// TIA Portal V21 export
FUNCTION_BLOCK "FB302"   // FB302, LAD
TITLE = FB302
{ S7_Optimized_Access := 'TRUE' }
AUTHOR : PRECISE
FAMILY : PRECISE
// MIXING
// stored: AutoNumber false, MemoryReserve 100, SetENOAutomatically false
   VAR_INPUT
      Enable : Bool;
      Disable : Bool;
      Fault : Bool;
      SecPulse : Bool;
      AlwaysTrue : Bool;
      StartConfirmationPopupSel : Bool;   // StartConfirmationPopupSel: 0-NO/1-YES
      EndConfirmationPopupSel : Bool;   // EndConfirmationPopupSel: 0-NO/1-YES
      MixingModeSel : Int;   // Mixing Mode Selection: 0-Auto/1-Manual
      MixerTypeSel : Int;   // Mixer Type Selection: 0-MM/1-USM/2-HSM/3-BP/4-ANCHOR
      MixingTimeBaseSel : Bool;   // Mixing Time Base Selection: 0-second/1-minute
      MixingTimeMin : Int := 1;   // For Mixing Mode Selection: 0-Auto & Mixing Time Base Selection: 1-minute
      MixingTimeSec : Int := 30;   // For Mixing Mode Selection: 0-Auto & Mixing Time Base Selection: 0-second
      MixingSpeed : Real := 100.0;
   END_VAR
   VAR_OUTPUT
      MixerCmd : Bool;
      WaterInletValve : Bool;
      StartConfirmationPopup : Bool;   // For Start Confirmation Popup Selection: Yes
      EndConfirmationPopup : Bool;   // For End Confirmation Popup Selection: Yes
      ManualPopup : Bool;   // For Mixing Mode Selection: 1-Manual
      MixingTimeMinPV : DInt;   // For Mixing Mode Selection: 0-Auto
      MixingTimeSecPV : DInt;   // For Mixing Mode Selection: 0-Auto
      MixingSpeedPV : Real;
      PrintTrigger : Bool;
      PrintWord : Int;
      PrintStatus : String[50];
   END_VAR
   VAR_IN_OUT
      Start : Bool;
      Stop : Bool;
      Reset : Bool;
      StartConfirmationAck : Bool;   // For Start Confirmation Popup Selection: Yes
      EndConfirmationAck : Bool;   // For End Confirmation Popup Selection: Yes
      ManualAck : Bool;   // For Mixing Mode Selection: 1-Manual
      Cp01Fsc : Bool;
      SpareBtn2 : Bool;
      Running : Bool;
      Selected : Bool;
      Paused : Bool;
      StartConfirmationPopupTemp : Bool;   // For Start Confirmation Popup Selection: Yes
      EndConfirmationPopupTemp : Bool;   // For End Confirmation Popup Selection: Yes
      ManualPopupTemp : Bool;   // For Mixing Mode Selection: 1-Manual
      MixingStarted : Bool;
      MixingOver : Bool;
   END_VAR
   VAR
      PrintTriggerTemp : Bool;
      RE1 : Bool;
      RE2 : Bool;
      RE3 : Bool;
      RE4 : Bool;
      RE5 : Bool;
      RE6 : Bool;
      RE7 : Bool;
      MixingTimer : "FB101";
      PrintTriggerResetTimer { S7_SetPoint := 'True'} : TON_TIME;
      BtnResetTimer { S7_SetPoint := 'True'} : TON_TIME;
   END_VAR
   VAR_TEMP
      STATUS1 : String[40];
      STATUS2 : String[40];
      STATUS3 : String[40];
      STATUS4 : String[40];
      STATUS5 : String[40];
   END_VAR
   VAR_TEMP   // added for the SCL form of the ladder/FBD networks
      _w1 : Bool;
      _w2 : Bool;
      _w3 : Bool;
      _w4 : Bool;
      _w5 : Bool;
   END_VAR
BEGIN

REGION Network 1: Running
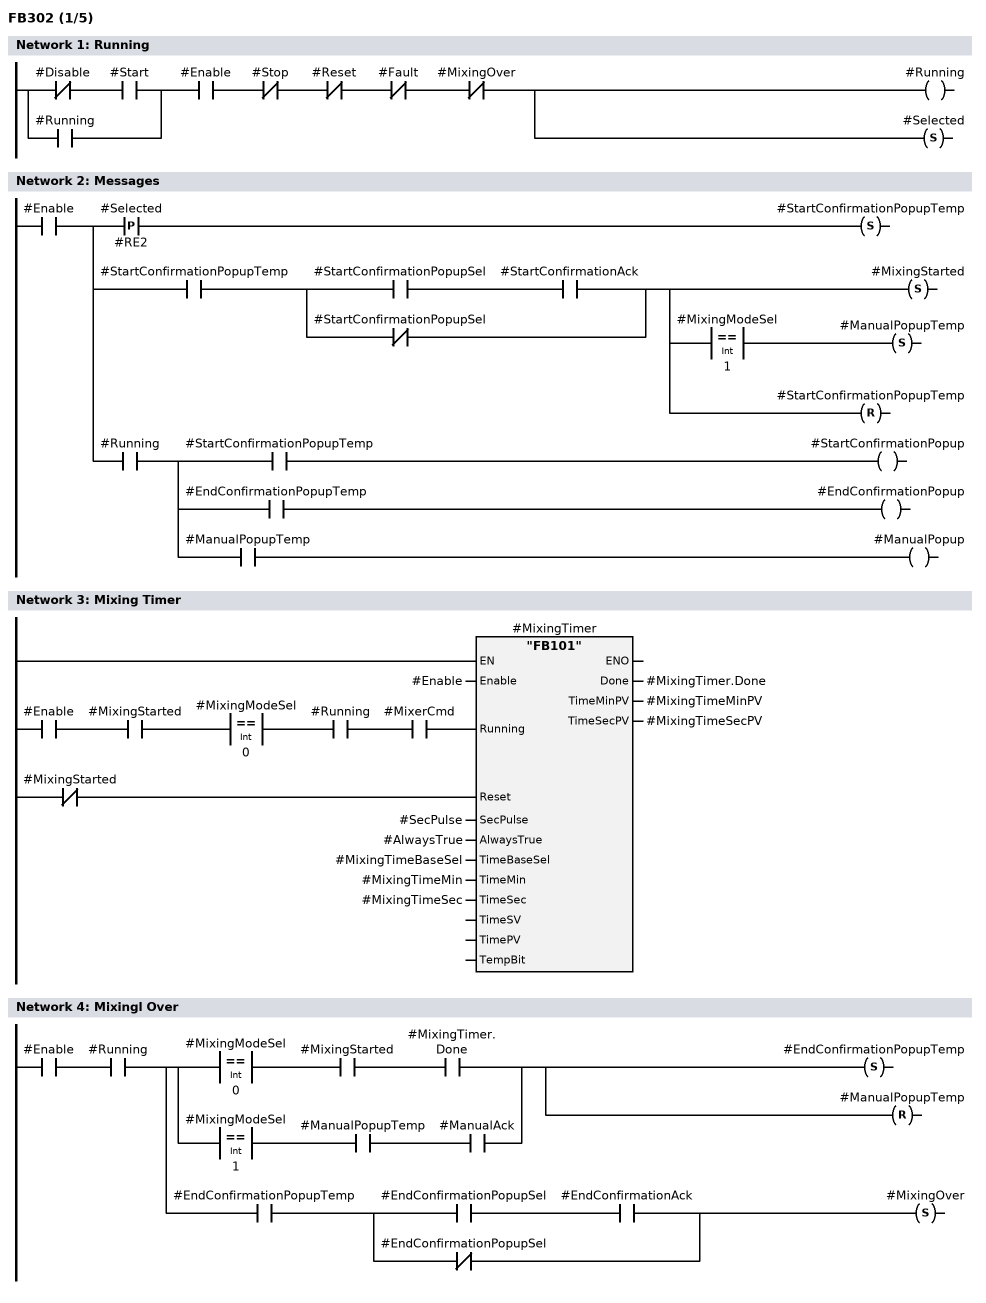
   RUNG wire#powerrail
      I_Contact( #Disable )
      Contact( #Start )
      wire#w1
      Contact( #Enable )
      I_Contact( #Stop )
      I_Contact( #Reset )
      I_Contact( #Fault )
      I_Contact( #MixingOver )
      wire#w2
      Coil( #Running )
   END_RUNG
   RUNG wire#powerrail
      Contact( #Running )
   END_RUNG wire#w1
   RUNG wire#w2
      S_Coil( #Selected )
   END_RUNG
   // the same network as SCL:
   #Running := ((NOT #Disable AND #Start) OR #Running) AND #Enable AND NOT #Stop AND NOT #Reset AND NOT #Fault AND NOT #MixingOver;
   IF #Running THEN #Selected := TRUE; END_IF;
END_REGION

REGION Network 2: Messages
   RUNG wire#powerrail
      Contact( #Enable )
      wire#w1
      P_Contact(operand := #Selected, bit := #RE2)
      S_Coil( #StartConfirmationPopupTemp )
   END_RUNG
   RUNG wire#w1
      Contact( #StartConfirmationPopupTemp )
      wire#w2
      Contact( #StartConfirmationPopupSel )
      Contact( #StartConfirmationAck )
      wire#w3
      S_Coil( #MixingStarted )
   END_RUNG
   RUNG wire#w2
      I_Contact( #StartConfirmationPopupSel )
   END_RUNG wire#w3
   RUNG wire#w3
      { S7_Templates := "SrcType := Int" } EQ_Contact(in1 := #MixingModeSel, in2 := 1)
      S_Coil( #ManualPopupTemp )
   END_RUNG
   RUNG wire#w3
      R_Coil( #StartConfirmationPopupTemp )
   END_RUNG
   RUNG wire#w1
      Contact( #Running )
      wire#w4
      Contact( #StartConfirmationPopupTemp )
      Coil( #StartConfirmationPopup )
   END_RUNG
   RUNG wire#w4
      Contact( #EndConfirmationPopupTemp )
      Coil( #EndConfirmationPopup )
   END_RUNG
   RUNG wire#w4
      Contact( #ManualPopupTemp )
      Coil( #ManualPopup )
   END_RUNG
   // the same network as SCL:
   #_w1 := #Enable AND #Selected AND NOT #RE2;   // rising edge of #Selected
   #RE2 := #Selected;
   IF #_w1 THEN #StartConfirmationPopupTemp := TRUE; END_IF;
   #_w2 := #Enable AND #StartConfirmationPopupTemp AND ((#StartConfirmationPopupSel AND #StartConfirmationAck) OR NOT #StartConfirmationPopupSel);
   IF #_w2 THEN #MixingStarted := TRUE; END_IF;
   IF #_w2 AND (#MixingModeSel = 1) THEN #ManualPopupTemp := TRUE; END_IF;
   IF #_w2 THEN #StartConfirmationPopupTemp := FALSE; END_IF;
   #_w3 := #Enable AND #Running;
   #StartConfirmationPopup := #_w3 AND #StartConfirmationPopupTemp;
   #EndConfirmationPopup := #_w3 AND #EndConfirmationPopupTemp;
   #ManualPopup := #_w3 AND #ManualPopupTemp;
END_REGION

REGION Network 3: Mixing Timer
   RUNG wire#powerrail
      #MixingTimer(Running := wire#w1, Reset := wire#w2, Enable := #Enable, SecPulse := #SecPulse, AlwaysTrue := #AlwaysTrue, TimeBaseSel := #MixingTimeBaseSel, TimeMin := #MixingTimeMin, TimeSec := #MixingTimeSec, TimeSV :=, TimePV :=, TempBit :=, Done => #MixingTimer.Done, TimeMinPV => #MixingTimeMinPV, TimeSecPV => #MixingTimeSecPV)
   END_RUNG
   RUNG wire#powerrail
      Contact( #Enable )
      Contact( #MixingStarted )
      { S7_Templates := "SrcType := Int" } EQ_Contact(in1 := #MixingModeSel, in2 := 0)
      Contact( #Running )
      Contact( #MixerCmd )
   END_RUNG wire#w1
   RUNG wire#powerrail
      I_Contact( #MixingStarted )
   END_RUNG wire#w2
   // the same network as SCL:
   #MixingTimer(Enable := #Enable,   // "FB101"
                Running := #Enable AND #MixingStarted AND (#MixingModeSel = 0) AND #Running AND #MixerCmd,
                Reset := NOT #MixingStarted,
                SecPulse := #SecPulse,
                AlwaysTrue := #AlwaysTrue,
                TimeBaseSel := #MixingTimeBaseSel,
                TimeMin := #MixingTimeMin,
                TimeSec := #MixingTimeSec,
                Done => #MixingTimer.Done,
                TimeMinPV => #MixingTimeMinPV,
                TimeSecPV => #MixingTimeSecPV);
END_REGION

REGION Network 4: Mixingl Over
   RUNG wire#powerrail
      Contact( #Enable )
      Contact( #Running )
      wire#w1
      { S7_Templates := "SrcType := Int" } EQ_Contact(in1 := #MixingModeSel, in2 := 0)
      Contact( #MixingStarted )
      Contact( #MixingTimer.Done )
      wire#w2
      S_Coil( #EndConfirmationPopupTemp )
   END_RUNG
   RUNG wire#w1
      { S7_Templates := "SrcType := Int" } EQ_Contact(in1 := #MixingModeSel, in2 := 1)
      Contact( #ManualPopupTemp )
      Contact( #ManualAck )
   END_RUNG wire#w2
   RUNG wire#w2
      R_Coil( #ManualPopupTemp )
   END_RUNG
   RUNG wire#w1
      Contact( #EndConfirmationPopupTemp )
      wire#w3
      Contact( #EndConfirmationPopupSel )
      Contact( #EndConfirmationAck )
      wire#w4
      S_Coil( #MixingOver )
   END_RUNG
   RUNG wire#w3
      I_Contact( #EndConfirmationPopupSel )
   END_RUNG wire#w4
   // the same network as SCL:
   #_w1 := #Enable AND #Running;
   IF #_w1 AND (((#MixingModeSel = 0) AND #MixingStarted AND #MixingTimer.Done) OR ((#MixingModeSel = 1) AND #ManualPopupTemp AND #ManualAck)) THEN
       #EndConfirmationPopupTemp := TRUE;
       #ManualPopupTemp := FALSE;
   END_IF;
   IF #_w1 AND #EndConfirmationPopupTemp AND ((#EndConfirmationPopupSel AND #EndConfirmationAck) OR NOT #EndConfirmationPopupSel) THEN
       #MixingOver := TRUE;
   END_IF;
END_REGION

REGION Network 5: Output On
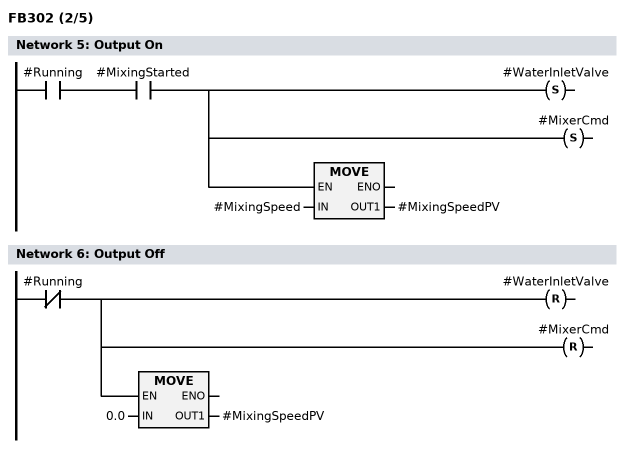
   RUNG wire#powerrail
      Contact( #Running )
      Contact( #MixingStarted )
      wire#w1
      S_Coil( #WaterInletValve )
   END_RUNG
   RUNG wire#w1
      S_Coil( #MixerCmd )
   END_RUNG
   RUNG wire#w1
      Move(in := #MixingSpeed, out1 => #MixingSpeedPV)
   END_RUNG
   // the same network as SCL:
   IF #Running AND #MixingStarted THEN
       #WaterInletValve := TRUE;
       #MixerCmd := TRUE;
       #MixingSpeedPV := #MixingSpeed;
   END_IF;
END_REGION

REGION Network 6: Output Off
   RUNG wire#powerrail
      I_Contact( #Running )
      wire#w1
      R_Coil( #WaterInletValve )
   END_RUNG
   RUNG wire#w1
      R_Coil( #MixerCmd )
   END_RUNG
   RUNG wire#w1
      Move(in := 0.0, out1 => #MixingSpeedPV)
   END_RUNG
   // the same network as SCL:
   IF NOT #Running THEN
       #WaterInletValve := FALSE;
       #MixerCmd := FALSE;
       #MixingSpeedPV := 0.0;
   END_IF;
END_REGION

REGION Network 7: Event Status
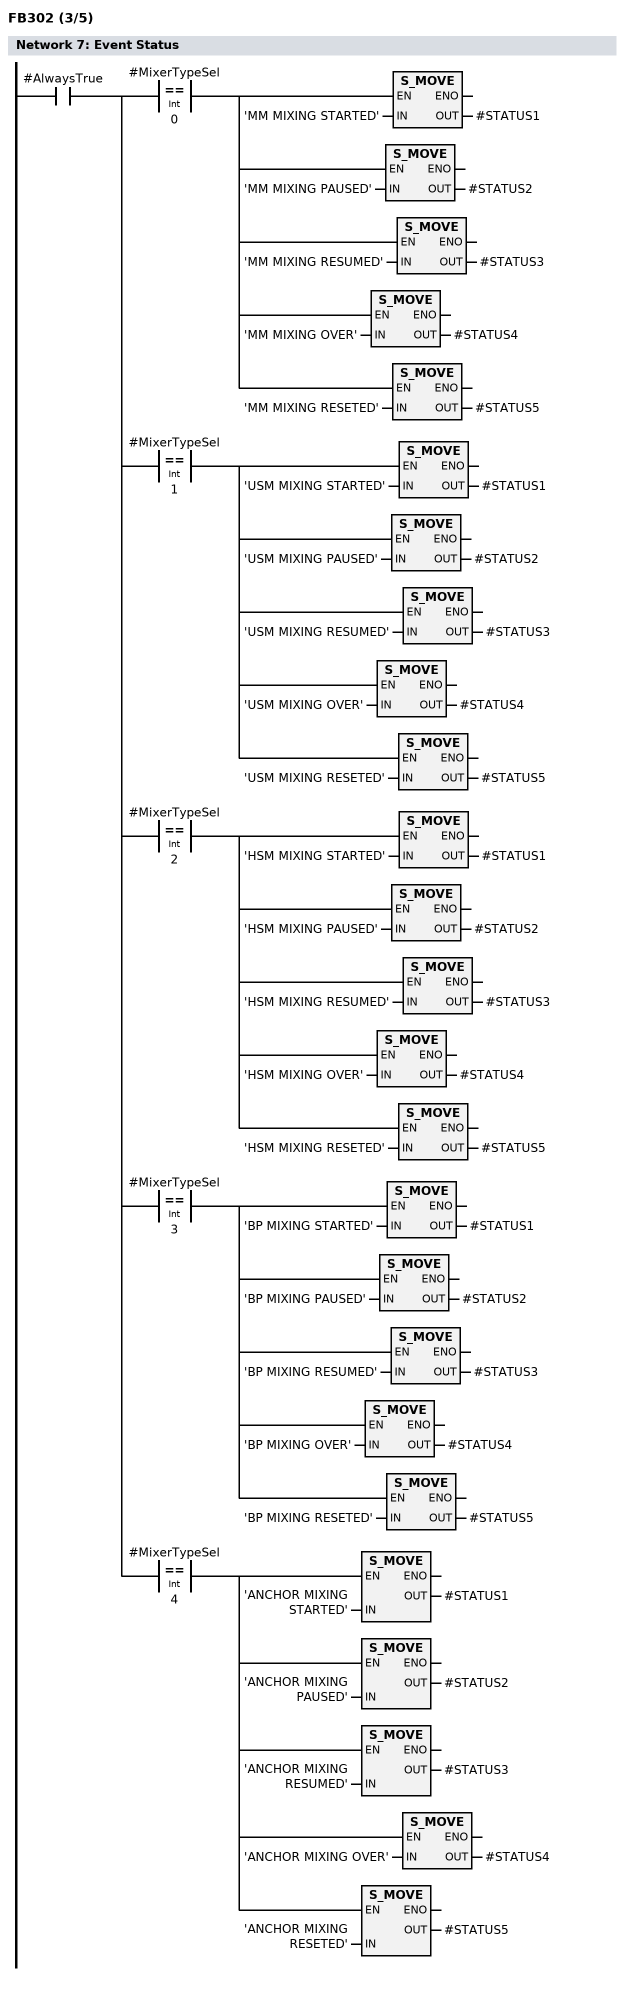
   RUNG wire#powerrail
      Contact( #AlwaysTrue )
      wire#w1
      { S7_Templates := "SrcType := Int" } EQ_Contact(in1 := #MixerTypeSel, in2 := 0)
      wire#w2
      S_Move(in := 'MM MIXING STARTED', out => #STATUS1)
   END_RUNG
   RUNG wire#w2
      S_Move(in := 'MM MIXING PAUSED', out => #STATUS2)
   END_RUNG
   RUNG wire#w2
      S_Move(in := 'MM MIXING RESUMED', out => #STATUS3)
   END_RUNG
   RUNG wire#w2
      S_Move(in := 'MM MIXING OVER', out => #STATUS4)
   END_RUNG
   RUNG wire#w2
      S_Move(in := 'MM MIXING RESETED', out => #STATUS5)
   END_RUNG
   RUNG wire#w1
      { S7_Templates := "SrcType := Int" } EQ_Contact(in1 := #MixerTypeSel, in2 := 1)
      wire#w3
      S_Move(in := 'USM MIXING STARTED', out => #STATUS1)
   END_RUNG
   RUNG wire#w3
      S_Move(in := 'USM MIXING PAUSED', out => #STATUS2)
   END_RUNG
   RUNG wire#w3
      S_Move(in := 'USM MIXING RESUMED', out => #STATUS3)
   END_RUNG
   RUNG wire#w3
      S_Move(in := 'USM MIXING OVER', out => #STATUS4)
   END_RUNG
   RUNG wire#w3
      S_Move(in := 'USM MIXING RESETED', out => #STATUS5)
   END_RUNG
   RUNG wire#w1
      { S7_Templates := "SrcType := Int" } EQ_Contact(in1 := #MixerTypeSel, in2 := 2)
      wire#w4
      S_Move(in := 'HSM MIXING STARTED', out => #STATUS1)
   END_RUNG
   RUNG wire#w4
      S_Move(in := 'HSM MIXING PAUSED', out => #STATUS2)
   END_RUNG
   RUNG wire#w4
      S_Move(in := 'HSM MIXING RESUMED', out => #STATUS3)
   END_RUNG
   RUNG wire#w4
      S_Move(in := 'HSM MIXING OVER', out => #STATUS4)
   END_RUNG
   RUNG wire#w4
      S_Move(in := 'HSM MIXING RESETED', out => #STATUS5)
   END_RUNG
   RUNG wire#w1
      { S7_Templates := "SrcType := Int" } EQ_Contact(in1 := #MixerTypeSel, in2 := 3)
      wire#w5
      S_Move(in := 'BP MIXING STARTED', out => #STATUS1)
   END_RUNG
   RUNG wire#w5
      S_Move(in := 'BP MIXING PAUSED', out => #STATUS2)
   END_RUNG
   RUNG wire#w5
      S_Move(in := 'BP MIXING RESUMED', out => #STATUS3)
   END_RUNG
   RUNG wire#w5
      S_Move(in := 'BP MIXING OVER', out => #STATUS4)
   END_RUNG
   RUNG wire#w5
      S_Move(in := 'BP MIXING RESETED', out => #STATUS5)
   END_RUNG
   RUNG wire#w1
      { S7_Templates := "SrcType := Int" } EQ_Contact(in1 := #MixerTypeSel, in2 := 4)
      wire#w6
      S_Move(in := 'ANCHOR MIXING STARTED', out => #STATUS1)
   END_RUNG
   RUNG wire#w6
      S_Move(in := 'ANCHOR MIXING PAUSED', out => #STATUS2)
   END_RUNG
   RUNG wire#w6
      S_Move(in := 'ANCHOR MIXING RESUMED', out => #STATUS3)
   END_RUNG
   RUNG wire#w6
      S_Move(in := 'ANCHOR MIXING OVER', out => #STATUS4)
   END_RUNG
   RUNG wire#w6
      S_Move(in := 'ANCHOR MIXING RESETED', out => #STATUS5)
   END_RUNG
   // the same network as SCL:
   IF #AlwaysTrue AND (#MixerTypeSel = 0) THEN
       #STATUS1 := 'MM MIXING STARTED';
       #STATUS2 := 'MM MIXING PAUSED';
       #STATUS3 := 'MM MIXING RESUMED';
       #STATUS4 := 'MM MIXING OVER';
       #STATUS5 := 'MM MIXING RESETED';
   END_IF;
   IF #AlwaysTrue AND (#MixerTypeSel = 1) THEN
       #STATUS1 := 'USM MIXING STARTED';
       #STATUS2 := 'USM MIXING PAUSED';
       #STATUS3 := 'USM MIXING RESUMED';
       #STATUS4 := 'USM MIXING OVER';
       #STATUS5 := 'USM MIXING RESETED';
   END_IF;
   IF #AlwaysTrue AND (#MixerTypeSel = 2) THEN
       #STATUS1 := 'HSM MIXING STARTED';
       #STATUS2 := 'HSM MIXING PAUSED';
       #STATUS3 := 'HSM MIXING RESUMED';
       #STATUS4 := 'HSM MIXING OVER';
       #STATUS5 := 'HSM MIXING RESETED';
   END_IF;
   IF #AlwaysTrue AND (#MixerTypeSel = 3) THEN
       #STATUS1 := 'BP MIXING STARTED';
       #STATUS2 := 'BP MIXING PAUSED';
       #STATUS3 := 'BP MIXING RESUMED';
       #STATUS4 := 'BP MIXING OVER';
       #STATUS5 := 'BP MIXING RESETED';
   END_IF;
   IF #AlwaysTrue AND (#MixerTypeSel = 4) THEN
       #STATUS1 := 'ANCHOR MIXING STARTED';
       #STATUS2 := 'ANCHOR MIXING PAUSED';
       #STATUS3 := 'ANCHOR MIXING RESUMED';
       #STATUS4 := 'ANCHOR MIXING OVER';
       #STATUS5 := 'ANCHOR MIXING RESETED';
   END_IF;
END_REGION

REGION Network 8: Print Logic
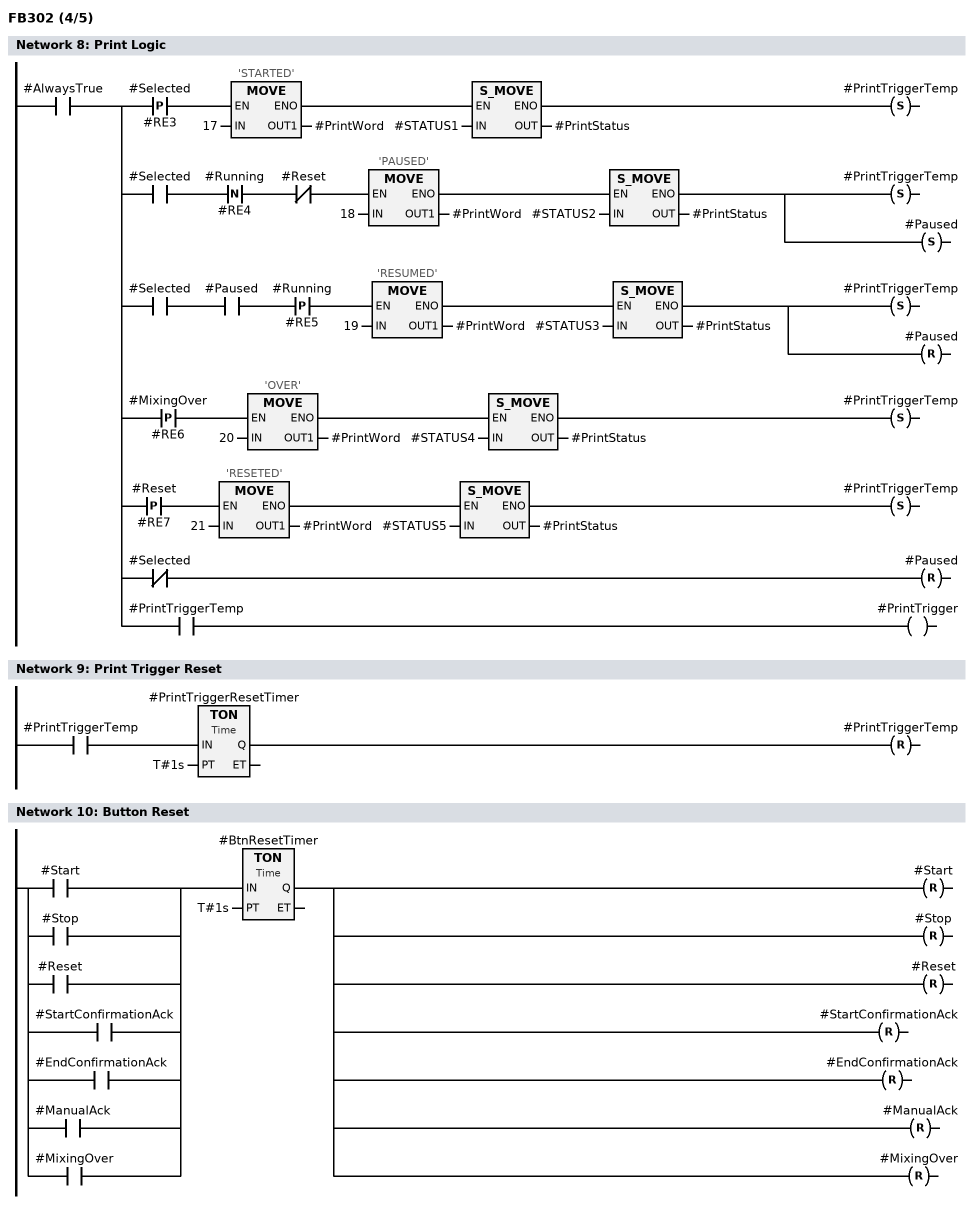
   RUNG wire#powerrail
      Contact( #AlwaysTrue )
      wire#w1
      P_Contact(operand := #Selected, bit := #RE3)
      { S7_GenerateENO := "TRUE" } Move(in := 17, out1 => #PrintWord)   // 'STARTED'
      S_Move(in := #STATUS1, out => #PrintStatus)
      S_Coil( #PrintTriggerTemp )
   END_RUNG
   RUNG wire#w1
      Contact( #Selected )
      N_Contact(operand := #Running, bit := #RE4)
      I_Contact( #Reset )
      { S7_GenerateENO := "TRUE" } Move(in := 18, out1 => #PrintWord)   // 'PAUSED'
      S_Move(in := #STATUS2, out => #PrintStatus)
      wire#w2
      S_Coil( #PrintTriggerTemp )
   END_RUNG
   RUNG wire#w2
      S_Coil( #Paused )
   END_RUNG
   RUNG wire#w1
      Contact( #Selected )
      Contact( #Paused )
      P_Contact(operand := #Running, bit := #RE5)
      { S7_GenerateENO := "TRUE" } Move(in := 19, out1 => #PrintWord)   // 'RESUMED'
      S_Move(in := #STATUS3, out => #PrintStatus)
      wire#w3
      S_Coil( #PrintTriggerTemp )
   END_RUNG
   RUNG wire#w3
      R_Coil( #Paused )
   END_RUNG
   RUNG wire#w1
      P_Contact(operand := #MixingOver, bit := #RE6)
      { S7_GenerateENO := "TRUE" } Move(in := 20, out1 => #PrintWord)   // 'OVER'
      S_Move(in := #STATUS4, out => #PrintStatus)
      S_Coil( #PrintTriggerTemp )
   END_RUNG
   RUNG wire#w1
      P_Contact(operand := #Reset, bit := #RE7)
      { S7_GenerateENO := "TRUE" } Move(in := 21, out1 => #PrintWord)   // 'RESETED'
      S_Move(in := #STATUS5, out => #PrintStatus)
      S_Coil( #PrintTriggerTemp )
   END_RUNG
   RUNG wire#w1
      I_Contact( #Selected )
      R_Coil( #Paused )
   END_RUNG
   RUNG wire#w1
      Contact( #PrintTriggerTemp )
      Coil( #PrintTrigger )
   END_RUNG
   // the same network as SCL:
   // ENO of a box is taken as its EN; it also drops when the box reports an error
   #_w1 := #AlwaysTrue AND #Selected AND NOT #RE3;   // rising edge of #Selected
   #RE3 := #Selected;
   IF #_w1 THEN
       #PrintWord := 17;   // 'STARTED'
       #PrintStatus := #STATUS1;
       #PrintTriggerTemp := TRUE;
   END_IF;
   #_w2 := #AlwaysTrue AND #Selected AND NOT #Running AND #RE4;   // falling edge of #Running
   #RE4 := #Running;
   IF #_w2 AND NOT #Reset THEN
       #PrintWord := 18;   // 'PAUSED'
       #PrintStatus := #STATUS2;
       #PrintTriggerTemp := TRUE;
       #Paused := TRUE;
   END_IF;
   #_w3 := #AlwaysTrue AND #Selected AND #Paused AND #Running AND NOT #RE5;   // rising edge of #Running
   #RE5 := #Running;
   IF #_w3 THEN
       #PrintWord := 19;   // 'RESUMED'
       #PrintStatus := #STATUS3;
       #PrintTriggerTemp := TRUE;
       #Paused := FALSE;
   END_IF;
   #_w4 := #AlwaysTrue AND #MixingOver AND NOT #RE6;   // rising edge of #MixingOver
   #RE6 := #MixingOver;
   IF #_w4 THEN
       #PrintWord := 20;   // 'OVER'
       #PrintStatus := #STATUS4;
       #PrintTriggerTemp := TRUE;
   END_IF;
   #_w5 := #AlwaysTrue AND #Reset AND NOT #RE7;   // rising edge of #Reset
   #RE7 := #Reset;
   IF #_w5 THEN
       #PrintWord := 21;   // 'RESETED'
       #PrintStatus := #STATUS5;
       #PrintTriggerTemp := TRUE;
   END_IF;
   IF #AlwaysTrue AND NOT #Selected THEN #Paused := FALSE; END_IF;
   #PrintTrigger := #AlwaysTrue AND #PrintTriggerTemp;
END_REGION

REGION Network 9: Print Trigger Reset
   RUNG wire#powerrail
      Contact( #PrintTriggerTemp )
      { S7_Templates := "time_type := Time" } #PrintTriggerResetTimer.TON(pt := T#1s, et =>)
      R_Coil( #PrintTriggerTemp )
   END_RUNG
   // the same network as SCL:
   #PrintTriggerResetTimer(IN := #PrintTriggerTemp, PT := T#1s);   // TON
   IF #PrintTriggerResetTimer.Q THEN #PrintTriggerTemp := FALSE; END_IF;
END_REGION

REGION Network 10: Button Reset
   RUNG wire#powerrail
      Contact( #Start )
      wire#w1
      { S7_Templates := "time_type := Time" } #BtnResetTimer.TON(pt := T#1s, et =>)
      wire#w2
      R_Coil( #Start )
   END_RUNG
   RUNG wire#powerrail
      Contact( #Stop )
   END_RUNG wire#w1
   RUNG wire#powerrail
      Contact( #Reset )
   END_RUNG wire#w1
   RUNG wire#powerrail
      Contact( #StartConfirmationAck )
   END_RUNG wire#w1
   RUNG wire#powerrail
      Contact( #EndConfirmationAck )
   END_RUNG wire#w1
   RUNG wire#powerrail
      Contact( #ManualAck )
   END_RUNG wire#w1
   RUNG wire#powerrail
      Contact( #MixingOver )
   END_RUNG wire#w1
   RUNG wire#w2
      R_Coil( #Stop )
   END_RUNG
   RUNG wire#w2
      R_Coil( #Reset )
   END_RUNG
   RUNG wire#w2
      R_Coil( #StartConfirmationAck )
   END_RUNG
   RUNG wire#w2
      R_Coil( #EndConfirmationAck )
   END_RUNG
   RUNG wire#w2
      R_Coil( #ManualAck )
   END_RUNG
   RUNG wire#w2
      R_Coil( #MixingOver )
   END_RUNG
   // the same network as SCL:
   #BtnResetTimer(IN := #Start OR #Stop OR #Reset OR #StartConfirmationAck OR #EndConfirmationAck OR #ManualAck OR #MixingOver,   // TON
                  PT := T#1s);
   IF #BtnResetTimer.Q THEN
       #Start := FALSE;
       #Stop := FALSE;
       #Reset := FALSE;
       #StartConfirmationAck := FALSE;
       #EndConfirmationAck := FALSE;
       #ManualAck := FALSE;
       #MixingOver := FALSE;
   END_IF;
END_REGION

REGION Network 11: Reset
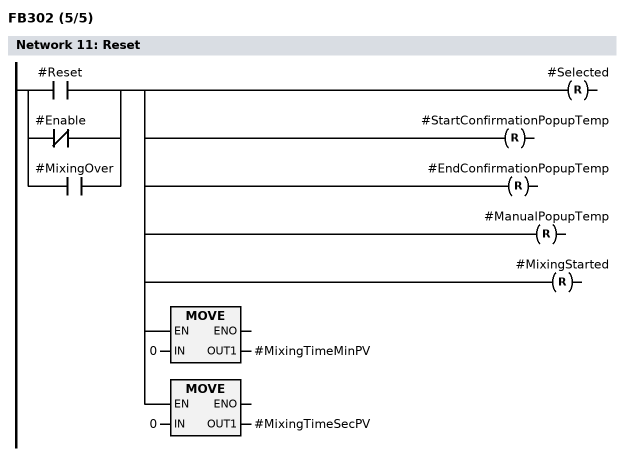
   RUNG wire#powerrail
      Contact( #Reset )
      wire#w1
      R_Coil( #Selected )
   END_RUNG
   RUNG wire#powerrail
      I_Contact( #Enable )
   END_RUNG wire#w1
   RUNG wire#powerrail
      Contact( #MixingOver )
   END_RUNG wire#w1
   RUNG wire#w1
      R_Coil( #StartConfirmationPopupTemp )
   END_RUNG
   RUNG wire#w1
      R_Coil( #EndConfirmationPopupTemp )
   END_RUNG
   RUNG wire#w1
      R_Coil( #ManualPopupTemp )
   END_RUNG
   RUNG wire#w1
      R_Coil( #MixingStarted )
   END_RUNG
   RUNG wire#w1
      { S7_GenerateENO := "TRUE" } Move(in := 0, out1 => #MixingTimeMinPV)
   END_RUNG
   RUNG wire#w1
      { S7_GenerateENO := "TRUE" } Move(in := 0, out1 => #MixingTimeSecPV)
   END_RUNG
   // the same network as SCL:
   IF #Reset OR NOT #Enable OR #MixingOver THEN
       #Selected := FALSE;
       #StartConfirmationPopupTemp := FALSE;
       #EndConfirmationPopupTemp := FALSE;
       #ManualPopupTemp := FALSE;
       #MixingStarted := FALSE;
       #MixingTimeMinPV := 0;
       #MixingTimeSecPV := 0;
   END_IF;
END_REGION
END_FUNCTION_BLOCK
